Omron CX-Programmer project NewProject (CX-Programmer 9.73)

# PLC NewPLC1: CP1L-E EM

## Global symbols (name address type ; comment)
0.00 BOOL  ; passo a passo formador fila entrada roler 41
0.01 BOOL  ; sensor peças maquineta descarga 41
0.02 BOOL  ; sensor sobre rolos entrada forno
0.03 BOOL  ; rele espaco forno 17 (saida 3.03)
0.04 BOOL  ; passo a passo formador fila entrada roler 42
0.05 BOOL  ; status roller desc. 42
0.06 BOOL  ; bancalino baixo carga forno 18
0.07 BOOL  ; rele forno 18 (saida 3.03)
0.08 BOOL  ; cnt de planos de carga 43
0.09 BOOL  ; cnt de planos de descarga 43
0.10 BOOL  ; bancalino entrada forno
0.11 BOOL  ; rele forno 22
1.00 BOOL  ; contagem de planos da carga carro
1.01 BOOL  ; status roller C41
1.02 BOOL  ; contador de gavetas carga roller mf42
1.03 BOOL  ; status roller C41
1.04 BOOL  ; contador descarga gaveta roller descarga mf42
1.05 BOOL  ; contagem de planos da descarga carro
1.08 BOOL  ; contagem peças roller carga 43
1.09 BOOL  ; status roller C43
1.11 BOOL  ; status roller D43
20.00 BOOL  ; reset retorno peças
20.01 BOOL  ; reset retorno peças
20.02 BOOL  ; reset retorno peças
30.02 BOOL  ; estoque vazio
30.04 BOOL  ; estoque zero mf42
30.05 BOOL  ; comparador planos  vazios
50.00 BOOL  ; liga cnt10
50.01 BOOL  ; reset cnt10
50.02 BOOL  ; liga cnt11
50.03 BOOL  ; reset cnt11
50.04 BOOL  ; liga cnt12
50.05 BOOL  ; reset cnt12
C0010 BOOL  ; reset inicio turno 1
C0011 BOOL  ; reset inicio turno 2
C0012 BOOL  ; reset inicio turno 3
C43 CHANNEL  ; contador de planos da 43
D1 CHANNEL  ; contador peças
D107 CHANNEL  ; peças por fila entrada forno
D205 CHANNEL  ; Segundos Relógio
D206 CHANNEL  ; Minutos Relógio
D207 CHANNEL  ; Horas Relogio
D208 CHANNEL  ; Dia Relógio
D209 CHANNEL  ; Mes Relogio
D210 CHANNEL  ; Ano Relogio
D211 CHANNEL  ; Ano Relogio 4 Digitos
D300 CHANNEL  ; Ano Relógio
D3001 CHANNEL  ; receita de destino RC43
D301 CHANNEL  ; Ano Relógio 4 digitos
D3800 CHANNEL  ; receita de destino F22
D400 CHANNEL  ; dia do mes
D402 CHANNEL  ; primeiro DM de contagem forno
D404 CHANNEL  ; peças por fila f17
D406 CHANNEL  ; peças por fila f18
D408 CHANNEL  ; peças por fila f22
D410 CHANNEL  ; primeiro DM envio roller
D500 CHANNEL  ; turno 1,2,3
D800 CHANNEL  ; horas
D802 CHANNEL  ; minutos
D804 CHANNEL  ; segundos
D806 CHANNEL  ; dia calendario
D808 CHANNEL  ; mês calendario
D810 CHANNEL  ; mês selecionado
D811 CHANNEL  ; linha selecionada
D910 CHANNEL  ; mês selecionado
H10.00 BOOL  ; forno com espaço
H10.01 BOOL  ; status roller carga 41
H10.02 BOOL  ; forno com espaço
H10.03 BOOL  ; roller carga 42
H10.04 BOOL  ; forno com espaço
H10.05 BOOL  ; status roller descarga 42
H10.06 BOOL  ; roller descarga 41
H10.07 BOOL  ; roller carga 43
H10.08 BOOL  ; status roller descarga 43
H19.15 BOOL  ; correção estoque IHM (mais)
H20.00 BOOL  ; Envia relogio superviório
H20.01 BOOL  ; correção estoque IHM (menos)
H20.02 BOOL  ; correção estoque IHM (menos)
H20.03 BOOL  ; correção estoque IHM (mais)
H20.04 BOOL  ; correção estoque IHM (menos)
H20.05 BOOL  ; correção estoque IHM (mais)
H20.06 BOOL  ; correcão estoque(menos)
H20.07 BOOL  ; correcão estoque(mais)
H20.08 BOOL  ; correcão estoque(menos)
H20.09 BOOL  ; correcão estoque(mais)
H20.10 BOOL  ; correcão estoque(menos)
H20.11 BOOL  ; correcão estoque(mais)
H30.00 BOOL  ; inicia contagem turno 1
H30.01 BOOL  ; inicia contagem turno 2
H30.02 BOOL  ; iniio contagem turno 3
T0001 BOOL  ; filtro senso
Banco_de_Dados Contador_de_Peças_RC43
Banco_de_Dados_ Contador_de_Peças_RC42
Banco_de_Dados_F17 Contador_de_Peças_F17
Banco_de_Dados_F18 Contador_de_Peças_F18
Banco_de_Dados_F22 Contador_de_Peças_F22
Banco_de_Dados_R42 Contador_de_Peças_RC42
Banco_de_Dados_R43 Contador_de_Peças_RC43
Banco_de_dados Contador_de_Peças_RC41
Banco_de_dados_R41 Contador_de_Peças_RC41
Reservado_1 D300 CHANNEL  ; reservado para elipse
Reservado_10 D309 CHANNEL  ; reservado para elipse
Reservado_11 D310 CHANNEL  ; reservado para elipse
Reservado_2 D301 CHANNEL  ; reservado para elipse
Reservado_3 D302 CHANNEL  ; reservado para elipse
Reservado_4 D303 CHANNEL  ; reservado para elipse
Reservado_5 D304 CHANNEL  ; reservado para elipse
Reservado_6 D305 CHANNEL  ; reservado para elipse
Reservado_7 D306 CHANNEL  ; reservado para elipse
Reservado_8 D307 CHANNEL  ; reservado para elipse
Reservado_9 D308 CHANNEL  ; reservado para elipse

## Program NewProgram1 (cyclic task 0)

### Section Principal

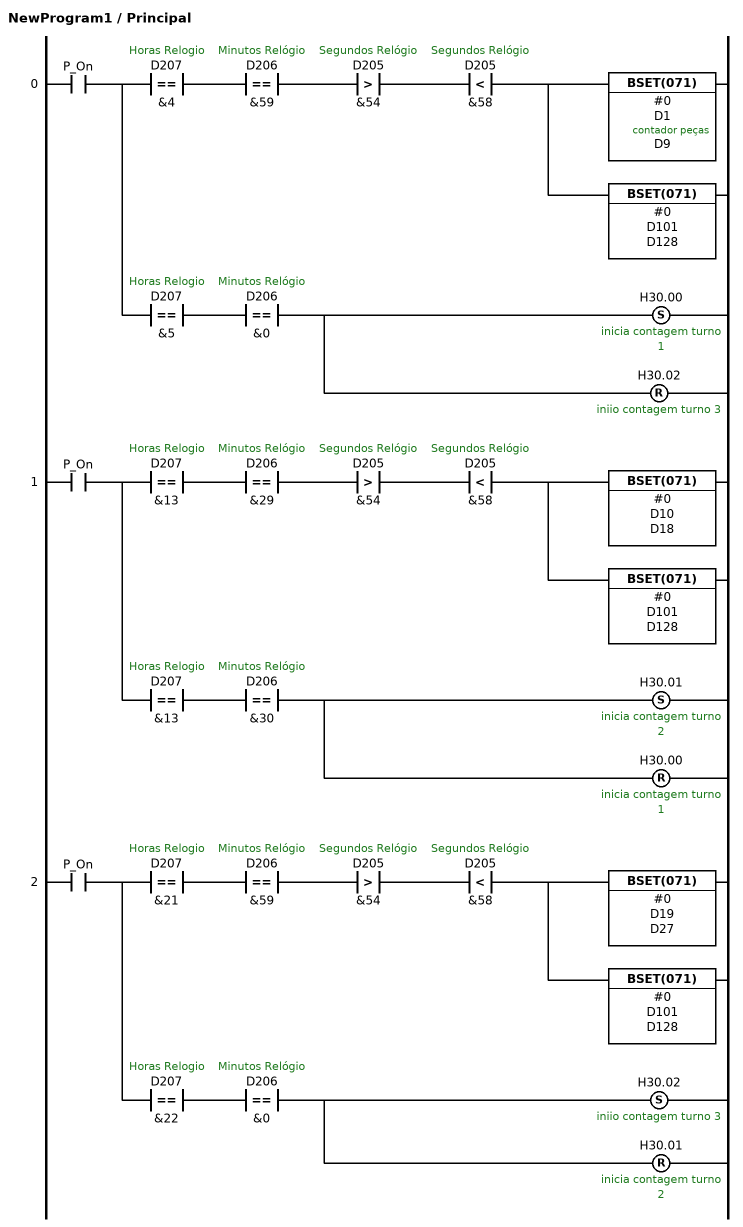
; rung 0
LD P_On
OUT TR0
AND=(300) D207 &4  ; Horas Relogio
AND=(300) D206 &59  ; Minutos Relógio
AND>(320) D205 &54  ; Segundos Relógio
AND<(310) D205 &58  ; Segundos Relógio
BSET(071) #0 D1 D9  ; contador peças
BSET(071) #0 D101 D128
LD TR0
AND=(300) D207 &5  ; Horas Relogio
AND=(300) D206 &0  ; Minutos Relógio
SET H30.00  ; inicia contagem turno 1
RSET H30.02  ; iniio contagem turno 3
; rung 1
LD P_On
OUT TR0
AND=(300) D207 &13  ; Horas Relogio
AND=(300) D206 &29  ; Minutos Relógio
AND>(320) D205 &54  ; Segundos Relógio
AND<(310) D205 &58  ; Segundos Relógio
BSET(071) #0 D10 D18
BSET(071) #0 D101 D128
LD TR0
AND=(300) D207 &13  ; Horas Relogio
AND=(300) D206 &30  ; Minutos Relógio
SET H30.01  ; inicia contagem turno 2
RSET H30.00  ; inicia contagem turno 1
; rung 2
LD P_On
OUT TR0
AND=(300) D207 &21  ; Horas Relogio
AND=(300) D206 &59  ; Minutos Relógio
AND>(320) D205 &54  ; Segundos Relógio
AND<(310) D205 &58  ; Segundos Relógio
BSET(071) #0 D19 D27
BSET(071) #0 D101 D128
LD TR0
AND=(300) D207 &22  ; Horas Relogio
AND=(300) D206 &0  ; Minutos Relógio
SET H30.02  ; iniio contagem turno 3
RSET H30.01  ; inicia contagem turno 2

### Section MF41

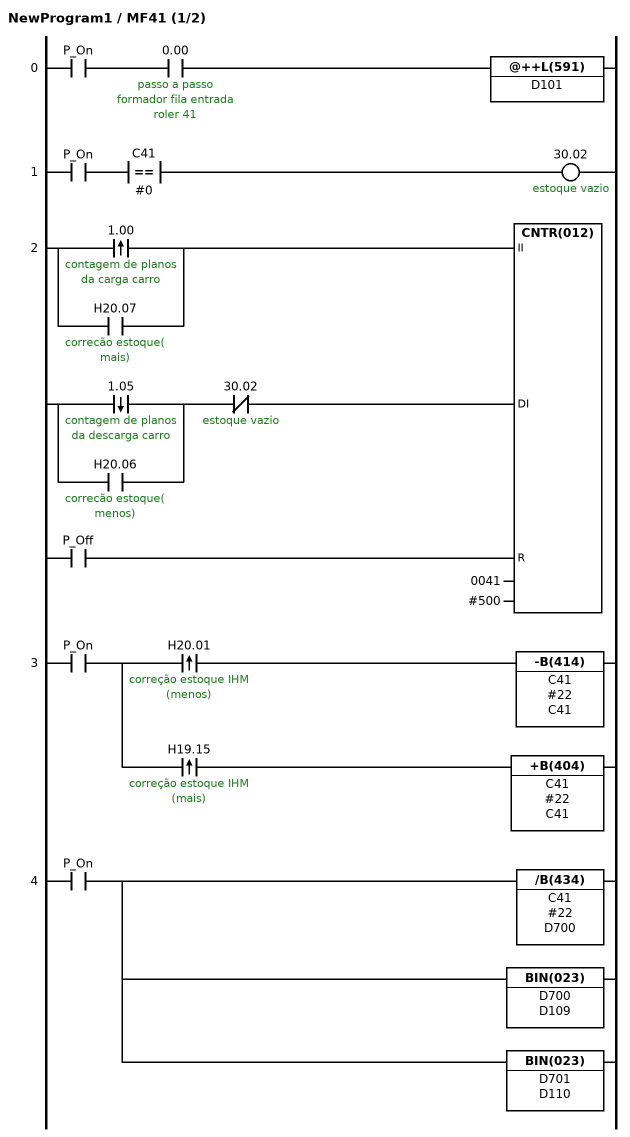
; rung 0
LD P_On
AND 0.00  ; passo a passo formador fila entrada roler 41
@++L(591) D101
; rung 1
LD P_On
AND=(300) C41 #0
OUT 30.02  ; estoque vazio
; rung 2
@LD 1.00  ; contagem de planos da carga carro
OR H20.07  ; correcão estoque(mais)
%LD 1.05  ; contagem de planos da descarga carro
OR H20.06  ; correcão estoque(menos)
ANDNOT 30.02  ; estoque vazio
LD P_Off
CNTR(012) 0041 #500
; rung 3
LD P_On
OUT TR0
@AND H20.01  ; correção estoque IHM (menos)
-B(414) C41 #22 C41
LD TR0
@AND H19.15  ; correção estoque IHM (mais)
+B(404) C41 #22 C41
; rung 4
LD P_On
/B(434) C41 #22 D700
BIN(023) D700 D109
BIN(023) D701 D110

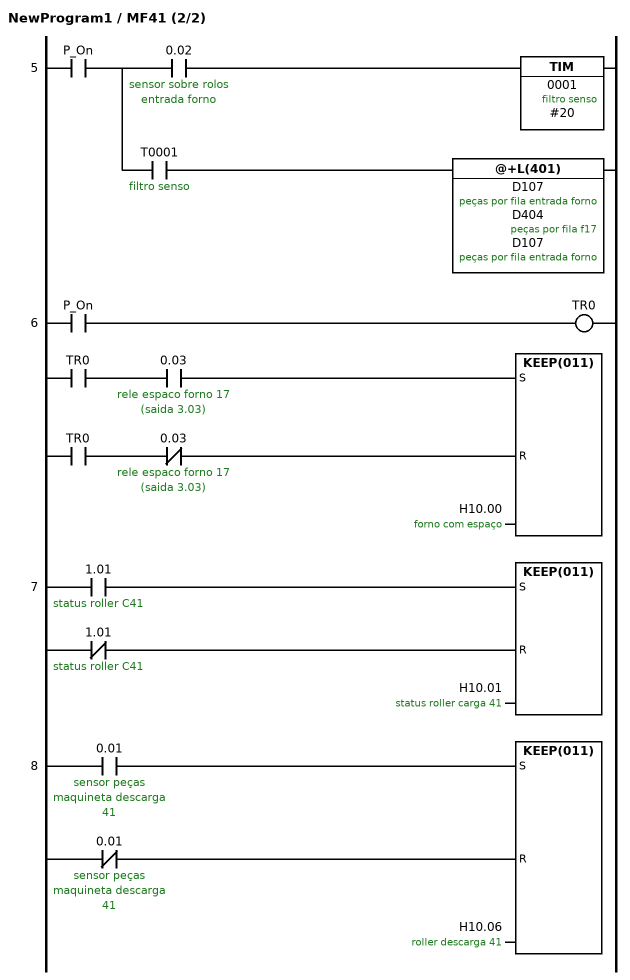
; rung 5
LD P_On
OUT TR0
AND 0.02  ; sensor sobre rolos entrada forno
TIM 0001 #20  ; filtro senso
LD TR0
AND T0001  ; filtro senso
@+L(401) D107 D404 D107  ; peças por fila entrada forno, peças por fila f17
; rung 6
LD P_On
OUT TR0
AND 0.03  ; rele espaco forno 17 (saida 3.03)
LD TR0
ANDNOT 0.03  ; rele espaco forno 17 (saida 3.03)
KEEP(011) H10.00  ; forno com espaço
; rung 7
LD 1.01  ; status roller C41
LDNOT 1.01  ; status roller C41
KEEP(011) H10.01  ; status roller carga 41
; rung 8
LD 0.01  ; sensor peças maquineta descarga 41
LDNOT 0.01  ; sensor peças maquineta descarga 41
KEEP(011) H10.06  ; roller descarga 41

### Section MF42

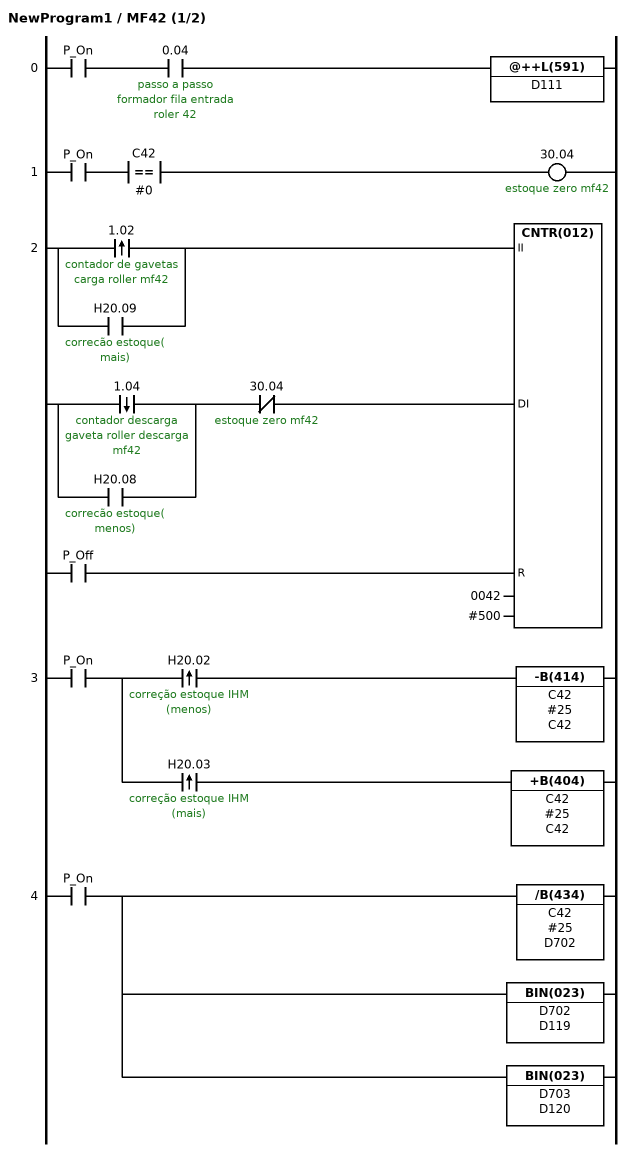
; rung 0
LD P_On
AND 0.04  ; passo a passo formador fila entrada roler 42
@++L(591) D111
; rung 1
LD P_On
AND=(300) C42 #0
OUT 30.04  ; estoque zero mf42
; rung 2
@LD 1.02  ; contador de gavetas carga roller mf42
OR H20.09  ; correcão estoque(mais)
%LD 1.04  ; contador descarga gaveta roller descarga mf42
OR H20.08  ; correcão estoque(menos)
ANDNOT 30.04  ; estoque zero mf42
LD P_Off
CNTR(012) 0042 #500
; rung 3
LD P_On
OUT TR0
@AND H20.02  ; correção estoque IHM (menos)
-B(414) C42 #25 C42
LD TR0
@AND H20.03  ; correção estoque IHM (mais)
+B(404) C42 #25 C42
; rung 4
LD P_On
/B(434) C42 #25 D702
BIN(023) D702 D119
BIN(023) D703 D120

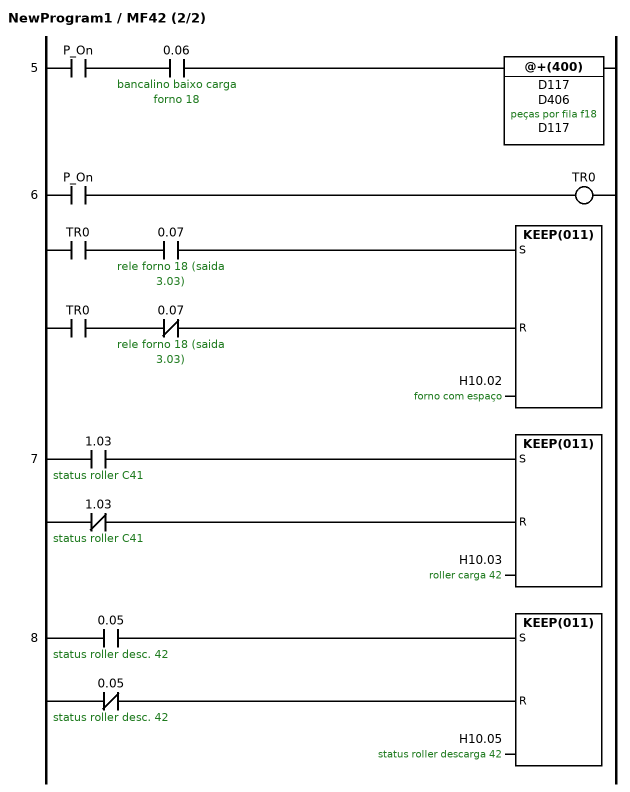
; rung 5
LD P_On
AND 0.06  ; bancalino baixo carga forno 18
@+(400) D117 D406 D117  ; peças por fila f18
; rung 6
LD P_On
OUT TR0
AND 0.07  ; rele forno 18 (saida 3.03)
LD TR0
ANDNOT 0.07  ; rele forno 18 (saida 3.03)
KEEP(011) H10.02  ; forno com espaço
; rung 7
LD 1.03  ; status roller C41
LDNOT 1.03  ; status roller C41
KEEP(011) H10.03  ; roller carga 42
; rung 8
LD 0.05  ; status roller desc. 42
LDNOT 0.05  ; status roller desc. 42
KEEP(011) H10.05  ; status roller descarga 42

### Section MF43

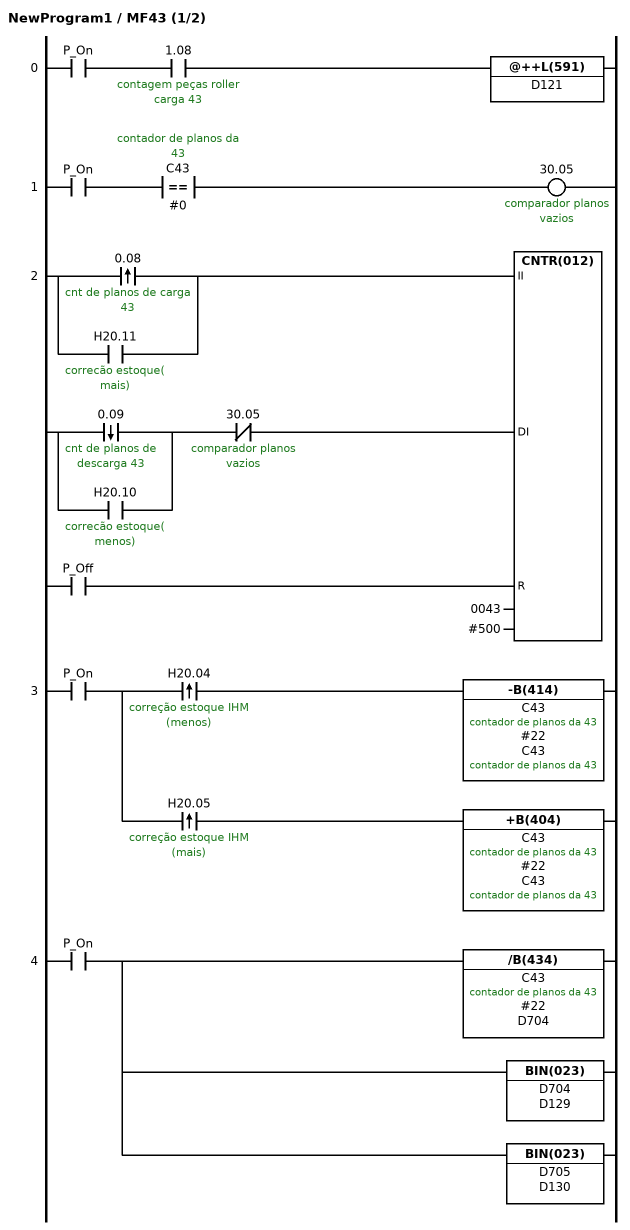
; rung 0
LD P_On
AND 1.08  ; contagem peças roller carga 43
@++L(591) D121
; rung 1
LD P_On
AND=(300) C43 #0  ; contador de planos da 43
OUT 30.05  ; comparador planos  vazios
; rung 2
@LD 0.08  ; cnt de planos de carga 43
OR H20.11  ; correcão estoque(mais)
%LD 0.09  ; cnt de planos de descarga 43
OR H20.10  ; correcão estoque(menos)
ANDNOT 30.05  ; comparador planos  vazios
LD P_Off
CNTR(012) 0043 #500
; rung 3
LD P_On
OUT TR0
@AND H20.04  ; correção estoque IHM (menos)
-B(414) C43 #22 C43  ; contador de planos da 43
LD TR0
@AND H20.05  ; correção estoque IHM (mais)
+B(404) C43 #22 C43  ; contador de planos da 43
; rung 4
LD P_On
/B(434) C43 #22 D704  ; contador de planos da 43
BIN(023) D704 D129
BIN(023) D705 D130

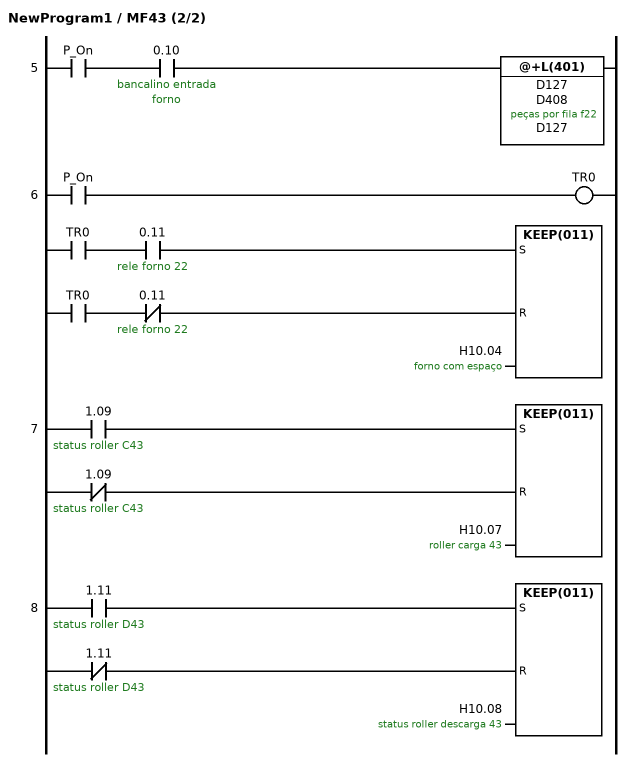
; rung 5
LD P_On
AND 0.10  ; bancalino entrada forno
@+L(401) D127 D408 D127  ; peças por fila f22
; rung 6
LD P_On
OUT TR0
AND 0.11  ; rele forno 22
LD TR0
ANDNOT 0.11  ; rele forno 22
KEEP(011) H10.04  ; forno com espaço
; rung 7
LD 1.09  ; status roller C43
LDNOT 1.09  ; status roller C43
KEEP(011) H10.07  ; roller carga 43
; rung 8
LD 1.11  ; status roller D43
LDNOT 1.11  ; status roller D43
KEEP(011) H10.08  ; status roller descarga 43

### Section MF41_ESPAÇO

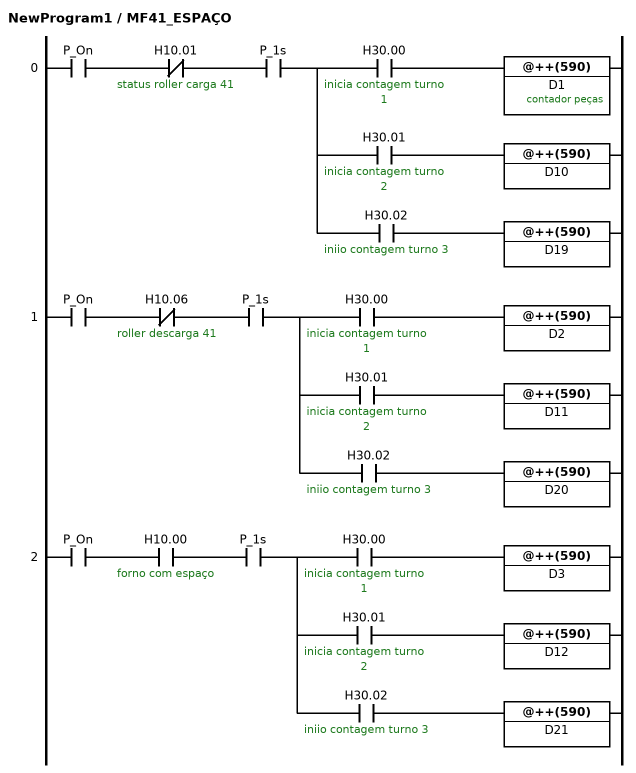
; rung 0
LD P_On
ANDNOT H10.01  ; status roller carga 41
AND P_1s
OUT TR0
AND H30.00  ; inicia contagem turno 1
@++(590) D1  ; contador peças  // 
LD TR0
AND H30.01  ; inicia contagem turno 2
@++(590) D10  // 
LD TR0
AND H30.02  ; iniio contagem turno 3
@++(590) D19  // 
; rung 1
LD P_On
ANDNOT H10.06  ; roller descarga 41
AND P_1s
OUT TR0
AND H30.00  ; inicia contagem turno 1
@++(590) D2  // 
LD TR0
AND H30.01  ; inicia contagem turno 2
@++(590) D11  // 
LD TR0
AND H30.02  ; iniio contagem turno 3
@++(590) D20  // 
; rung 2
LD P_On
AND H10.00  ; forno com espaço
AND P_1s
OUT TR0
AND H30.00  ; inicia contagem turno 1
@++(590) D3  // 
LD TR0
AND H30.01  ; inicia contagem turno 2
@++(590) D12  // 
LD TR0
AND H30.02  ; iniio contagem turno 3
@++(590) D21  // 

### Section MF42_ESPAÇO

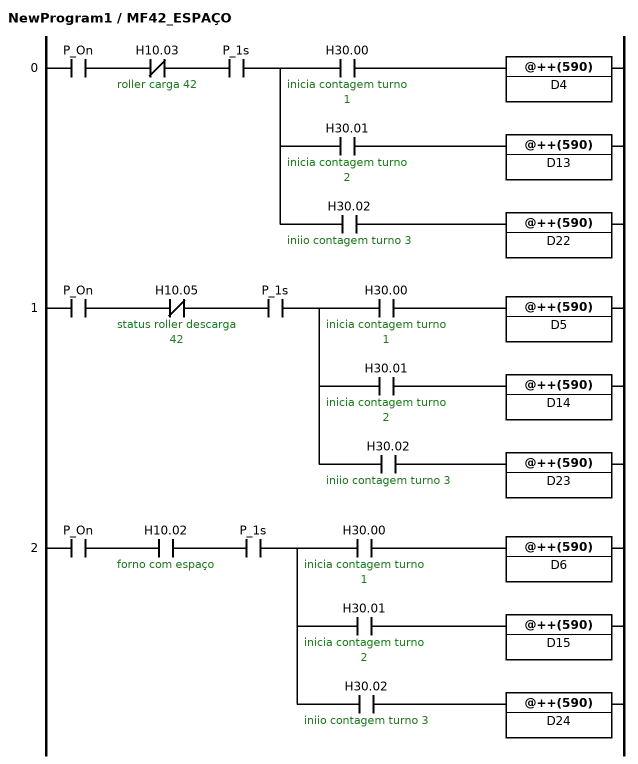
; rung 0
LD P_On
ANDNOT H10.03  ; roller carga 42
AND P_1s
OUT TR0
AND H30.00  ; inicia contagem turno 1
@++(590) D4  // 
LD TR0
AND H30.01  ; inicia contagem turno 2
@++(590) D13  // 
LD TR0
AND H30.02  ; iniio contagem turno 3
@++(590) D22  // 
; rung 1
LD P_On
ANDNOT H10.05  ; status roller descarga 42
AND P_1s
OUT TR0
AND H30.00  ; inicia contagem turno 1
@++(590) D5  // 
LD TR0
AND H30.01  ; inicia contagem turno 2
@++(590) D14  // 
LD TR0
AND H30.02  ; iniio contagem turno 3
@++(590) D23  // 
; rung 2
LD P_On
AND H10.02  ; forno com espaço
AND P_1s
OUT TR0
AND H30.00  ; inicia contagem turno 1
@++(590) D6  // 
LD TR0
AND H30.01  ; inicia contagem turno 2
@++(590) D15  // 
LD TR0
AND H30.02  ; iniio contagem turno 3
@++(590) D24  // 

### Section MF43_ESPAÇO

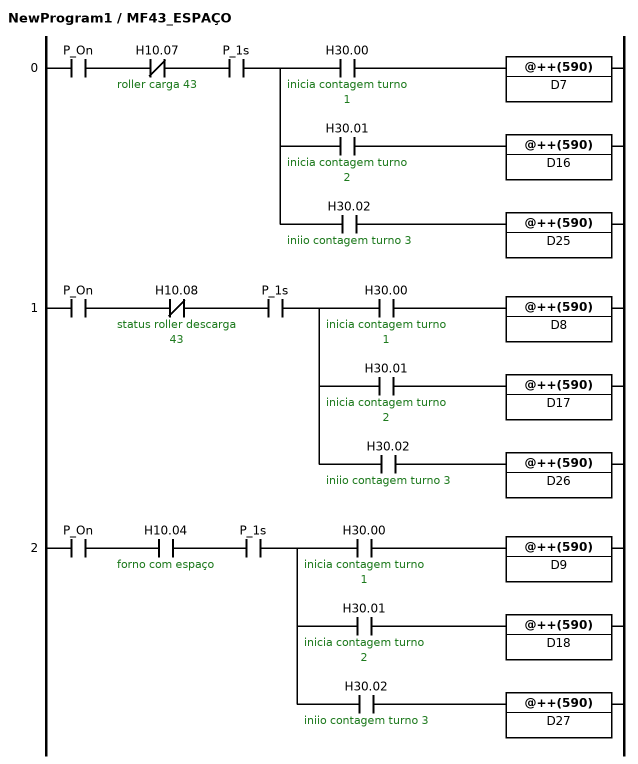
; rung 0
LD P_On
ANDNOT H10.07  ; roller carga 43
AND P_1s
OUT TR0
AND H30.00  ; inicia contagem turno 1
@++(590) D7  // 
LD TR0
AND H30.01  ; inicia contagem turno 2
@++(590) D16  // 
LD TR0
AND H30.02  ; iniio contagem turno 3
@++(590) D25  // 
; rung 1
LD P_On
ANDNOT H10.08  ; status roller descarga 43
AND P_1s
OUT TR0
AND H30.00  ; inicia contagem turno 1
@++(590) D8  // 
LD TR0
AND H30.01  ; inicia contagem turno 2
@++(590) D17  // 
LD TR0
AND H30.02  ; iniio contagem turno 3
@++(590) D26  // 
; rung 2
LD P_On
AND H10.04  ; forno com espaço
AND P_1s
OUT TR0
AND H30.00  ; inicia contagem turno 1
@++(590) D9  // 
LD TR0
AND H30.01  ; inicia contagem turno 2
@++(590) D18  // 
LD TR0
AND H30.02  ; iniio contagem turno 3
@++(590) D27  // 

### Section Banco_de_Dados

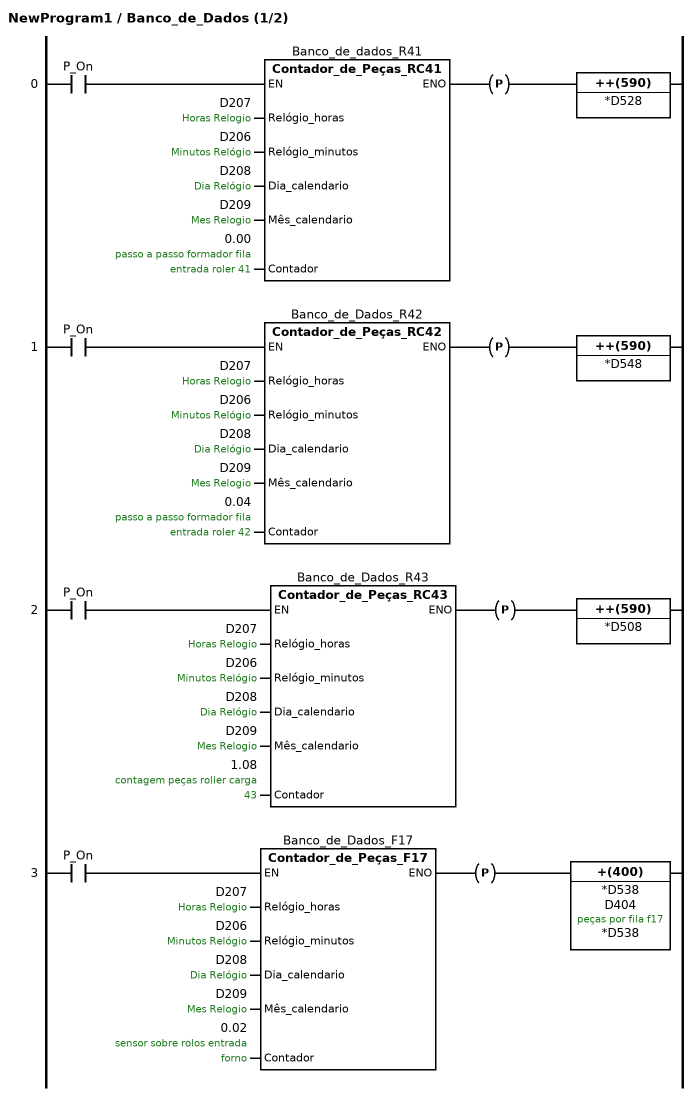
; rung 0
LD P_On
CALL Banco_de_dados_R41 : Contador_de_Peças_RC41 (Relógio_horas := D207, Relógio_minutos := D206, Dia_calendario := D208, Mês_calendario := D209, Contador := 0.00)  ; Horas Relogio, Minutos Relógio, Dia Relógio, Mes Relogio, passo a passo formador fila entrada roler 41
UP(521)
++(590) *D528
; rung 1
LD P_On
CALL Banco_de_Dados_R42 : Contador_de_Peças_RC42 (Relógio_horas := D207, Relógio_minutos := D206, Dia_calendario := D208, Mês_calendario := D209, Contador := 0.04)  ; Horas Relogio, Minutos Relógio, Dia Relógio, Mes Relogio, passo a passo formador fila entrada roler 42
UP(521)
++(590) *D548
; rung 2
LD P_On
CALL Banco_de_Dados_R43 : Contador_de_Peças_RC43 (Relógio_horas := D207, Relógio_minutos := D206, Dia_calendario := D208, Mês_calendario := D209, Contador := 1.08)  ; Horas Relogio, Minutos Relógio, Dia Relógio, Mes Relogio, contagem peças roller carga 43
UP(521)
++(590) *D508
; rung 3
LD P_On
CALL Banco_de_Dados_F17 : Contador_de_Peças_F17 (Relógio_horas := D207, Relógio_minutos := D206, Dia_calendario := D208, Mês_calendario := D209, Contador := 0.02)  ; Horas Relogio, Minutos Relógio, Dia Relógio, Mes Relogio, sensor sobre rolos entrada forno
UP(521)
+(400) *D538 D404 *D538  ; peças por fila f17

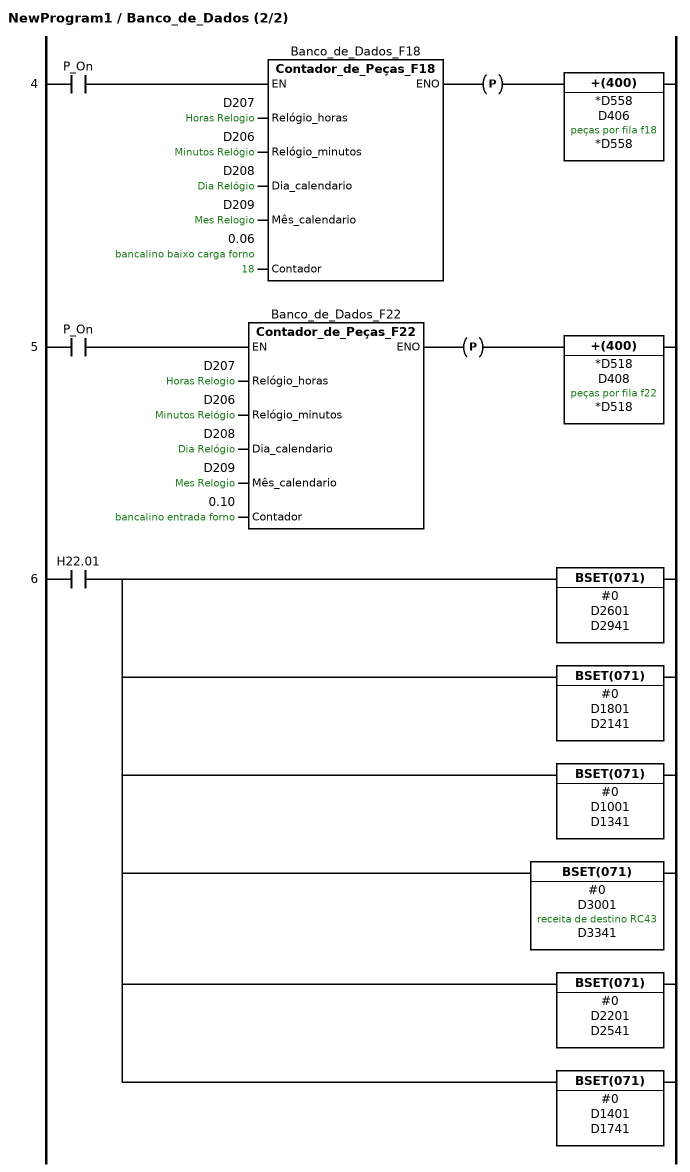
; rung 4
LD P_On
CALL Banco_de_Dados_F18 : Contador_de_Peças_F18 (Relógio_horas := D207, Relógio_minutos := D206, Dia_calendario := D208, Mês_calendario := D209, Contador := 0.06)  ; Horas Relogio, Minutos Relógio, Dia Relógio, Mes Relogio, bancalino baixo carga forno 18
UP(521)
+(400) *D558 D406 *D558  ; peças por fila f18
; rung 5
LD P_On
CALL Banco_de_Dados_F22 : Contador_de_Peças_F22 (Relógio_horas := D207, Relógio_minutos := D206, Dia_calendario := D208, Mês_calendario := D209, Contador := 0.10)  ; Horas Relogio, Minutos Relógio, Dia Relógio, Mes Relogio, bancalino entrada forno
UP(521)
+(400) *D518 D408 *D518  ; peças por fila f22
; rung 6
LD H22.01
BSET(071) #0 D2601 D2941
BSET(071) #0 D1801 D2141
BSET(071) #0 D1001 D1341
BSET(071) #0 D3001 D3341  ; receita de destino RC43
BSET(071) #0 D2201 D2541
BSET(071) #0 D1401 D1741

### Section Transferencia_excel

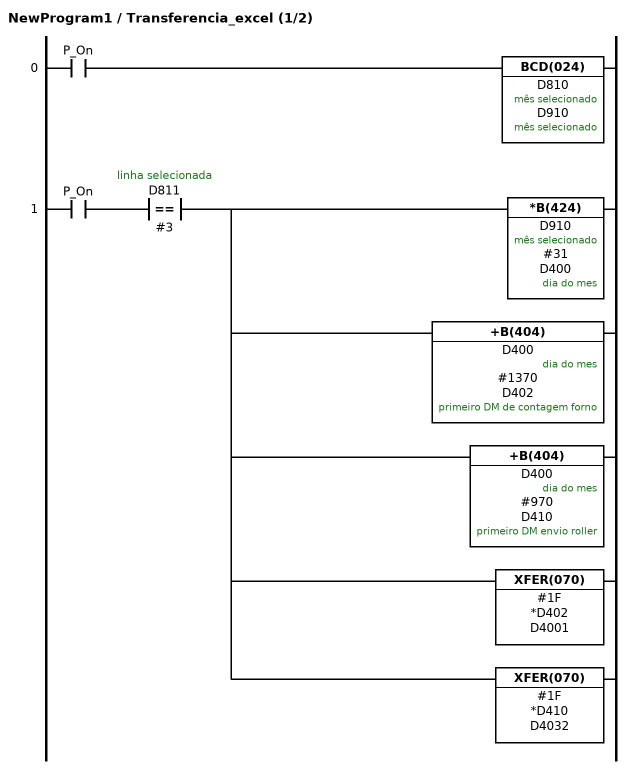
; rung 0
LD P_On
BCD(024) D810 D910  ; mês selecionado
; rung 1
LD P_On
AND=(300) D811 #3  ; linha selecionada
*B(424) D910 #31 D400  ; mês selecionado, dia do mes
+B(404) D400 #1370 D402  ; dia do mes, primeiro DM de contagem forno
+B(404) D400 #970 D410  ; dia do mes, primeiro DM envio roller
XFER(070) #1F *D402 D4001
XFER(070) #1F *D410 D4032

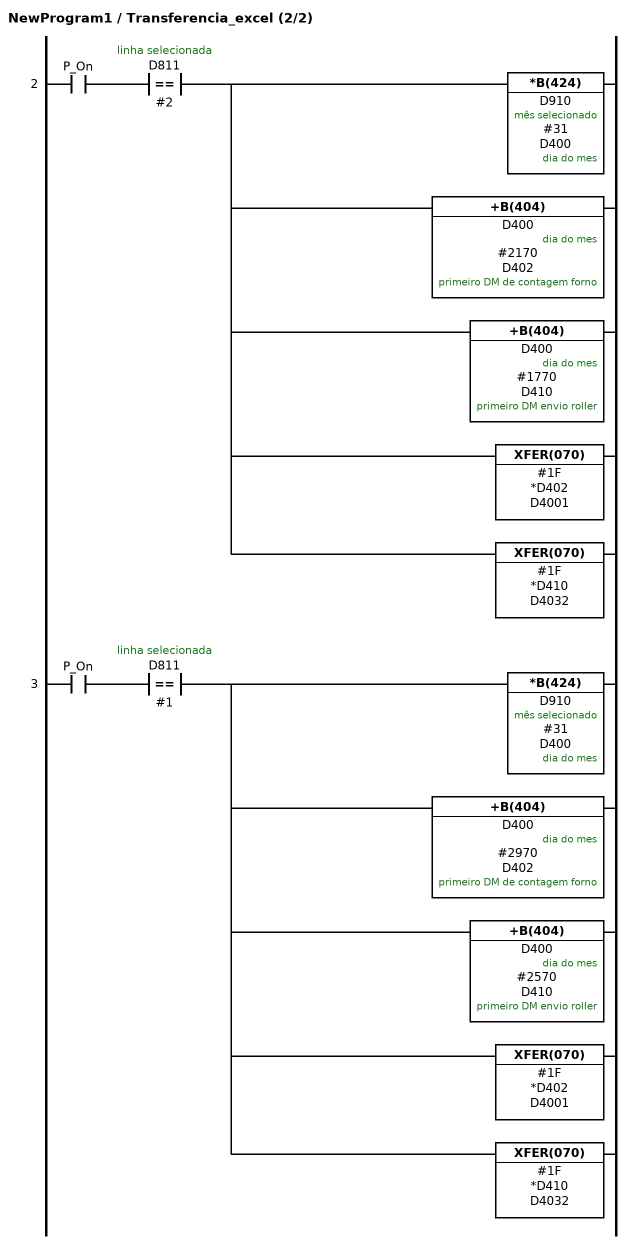
; rung 2
LD P_On
AND=(300) D811 #2  ; linha selecionada
*B(424) D910 #31 D400  ; mês selecionado, dia do mes
+B(404) D400 #2170 D402  ; dia do mes, primeiro DM de contagem forno
+B(404) D400 #1770 D410  ; dia do mes, primeiro DM envio roller
XFER(070) #1F *D402 D4001
XFER(070) #1F *D410 D4032
; rung 3
LD P_On
AND=(300) D811 #1  ; linha selecionada
*B(424) D910 #31 D400  ; mês selecionado, dia do mes
+B(404) D400 #2970 D402  ; dia do mes, primeiro DM de contagem forno
+B(404) D400 #2570 D410  ; dia do mes, primeiro DM envio roller
XFER(070) #1F *D402 D4001
XFER(070) #1F *D410 D4032

### Section Relogio

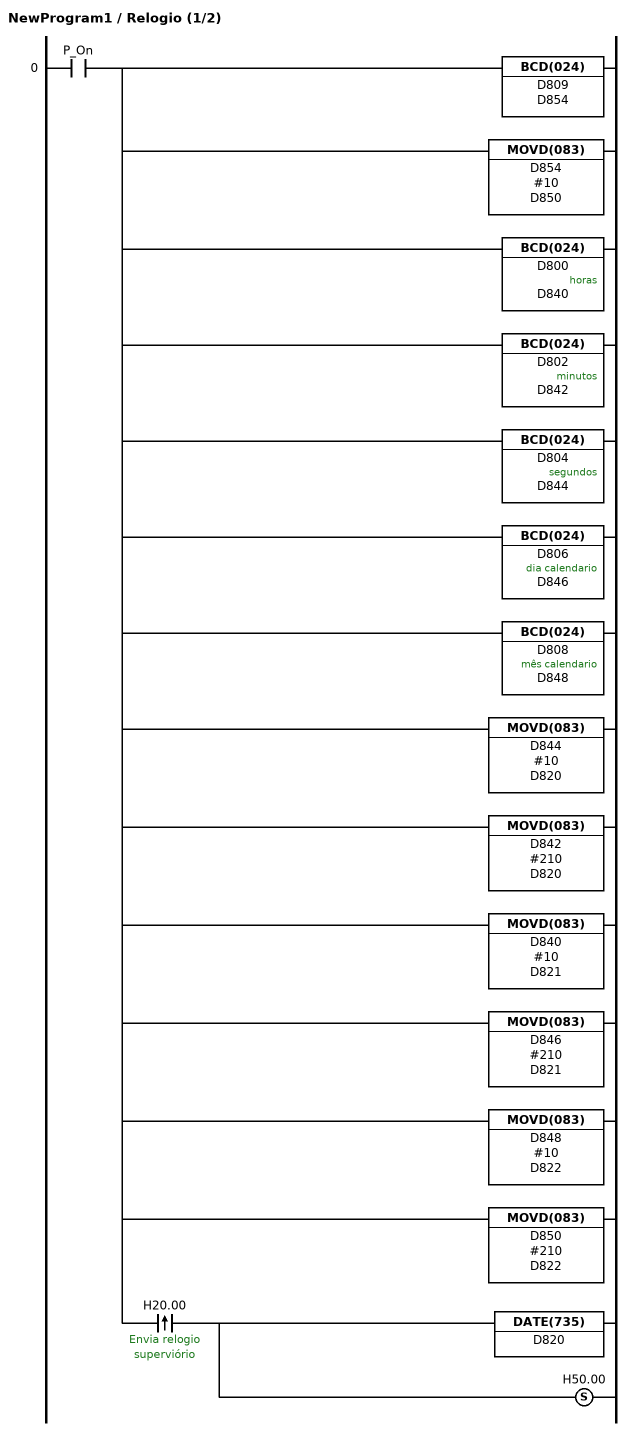
; rung 0
LD P_On
BCD(024) D809 D854
MOVD(083) D854 #10 D850
BCD(024) D800 D840  ; horas
BCD(024) D802 D842  ; minutos
BCD(024) D804 D844  ; segundos
BCD(024) D806 D846  ; dia calendario
BCD(024) D808 D848  ; mês calendario
MOVD(083) D844 #10 D820
MOVD(083) D842 #210 D820
MOVD(083) D840 #10 D821
MOVD(083) D846 #210 D821
MOVD(083) D848 #10 D822
MOVD(083) D850 #210 D822
@AND H20.00  ; Envia relogio superviório
DATE(735) D820
SET H50.00

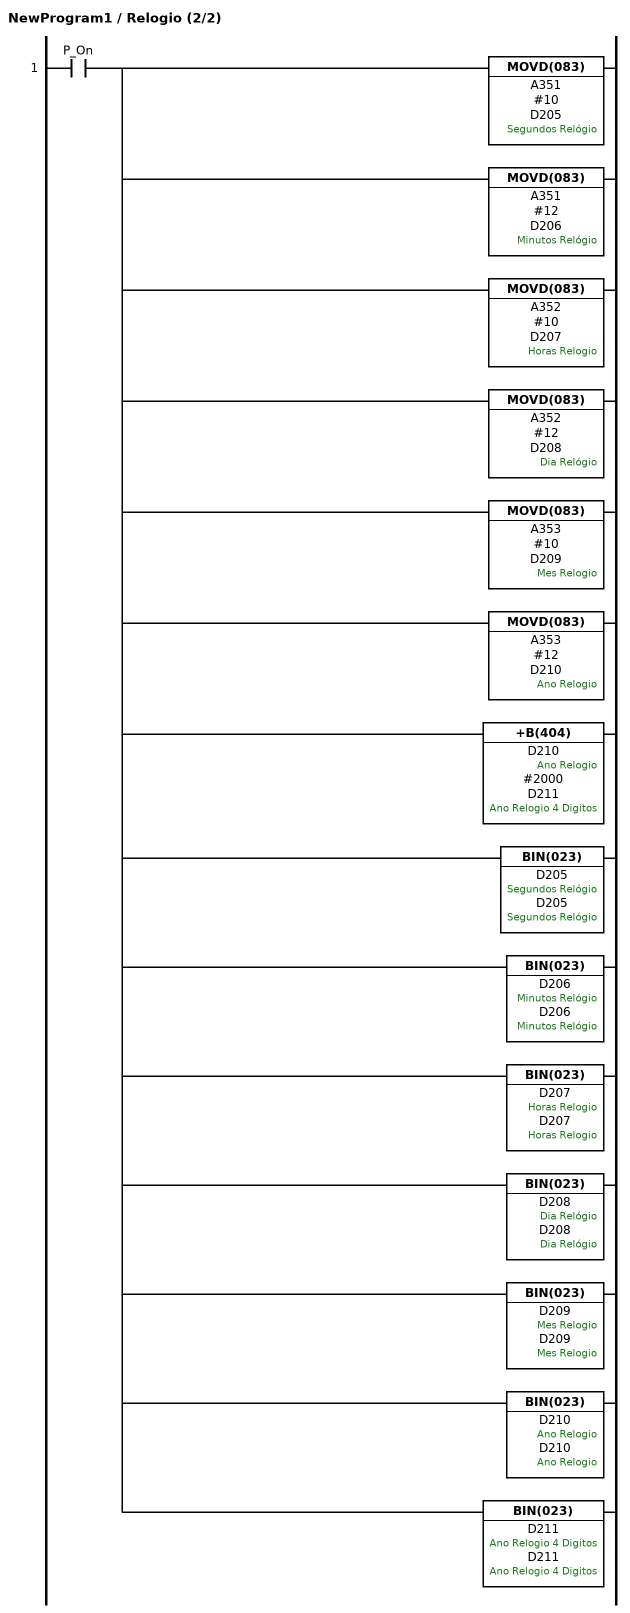
; rung 1
LD P_On
MOVD(083) A351 #10 D205  ; Segundos Relógio
MOVD(083) A351 #12 D206  ; Minutos Relógio
MOVD(083) A352 #10 D207  ; Horas Relogio
MOVD(083) A352 #12 D208  ; Dia Relógio
MOVD(083) A353 #10 D209  ; Mes Relogio
MOVD(083) A353 #12 D210  ; Ano Relogio
+B(404) D210 #2000 D211  ; Ano Relogio, Ano Relogio 4 Digitos
BIN(023) D205 D205  ; Segundos Relógio
BIN(023) D206 D206  ; Minutos Relógio
BIN(023) D207 D207  ; Horas Relogio
BIN(023) D208 D208  ; Dia Relógio
BIN(023) D209 D209  ; Mes Relogio
BIN(023) D210 D210  ; Ano Relogio
BIN(023) D211 D211  ; Ano Relogio 4 Digitos

### Section End
; rung 0
END(001)

## Function block Contador_de_Peças_F17
VAR_INPUT
  Relógio_horas : WORD;
  Relógio_minutos : WORD;
  Dia_calendario : WORD;
  Mês_calendario : WORD;
  Contador : BOOL;
END_VAR
VAR
  _31dias_vezes_2 AT D530 : WORD;
  Ponteiro_DWord AT D532 : WORD;
  Memória_de_Armazenagem AT D534 : WORD;
  Memoria_contagem_BIN AT D536 : WORD;
  Memoria_contagem_BCD AT D538 : WORD;
END_VAR

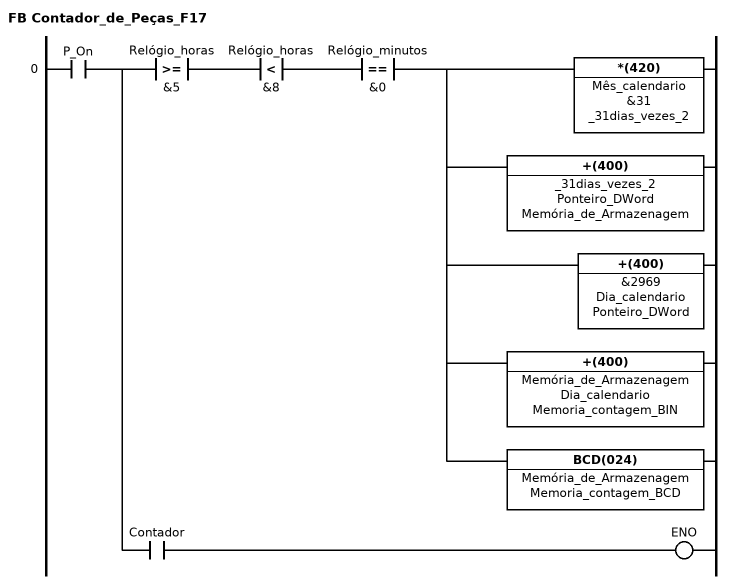
; rung 0
LD P_On
OUT TR0
AND>=(325) Relógio_horas &5
AND<(310) Relógio_horas &8
AND=(300) Relógio_minutos &0
*(420) Mês_calendario &31 _31dias_vezes_2
+(400) _31dias_vezes_2 Ponteiro_DWord Memória_de_Armazenagem
+(400) &2969 Dia_calendario Ponteiro_DWord
+(400) Memória_de_Armazenagem Dia_calendario Memoria_contagem_BIN
BCD(024) Memória_de_Armazenagem Memoria_contagem_BCD
LD TR0
AND Contador
OUT ENO

## Function block Contador_de_Peças_F18
VAR_INPUT
  Relógio_horas : WORD;
  Relógio_minutos : WORD;
  Dia_calendario : WORD;
  Mês_calendario : WORD;
  Contador : BOOL;
END_VAR
VAR
  _31dias_vezes_2 AT D550 : WORD;
  Ponteiro_DWord AT D552 : WORD;
  Memória_de_Armazenagem AT D554 : WORD;
  Memoria_contagem_BIN AT D556 : WORD;
  Memoria_contagem_BCD AT D558 : WORD;
END_VAR

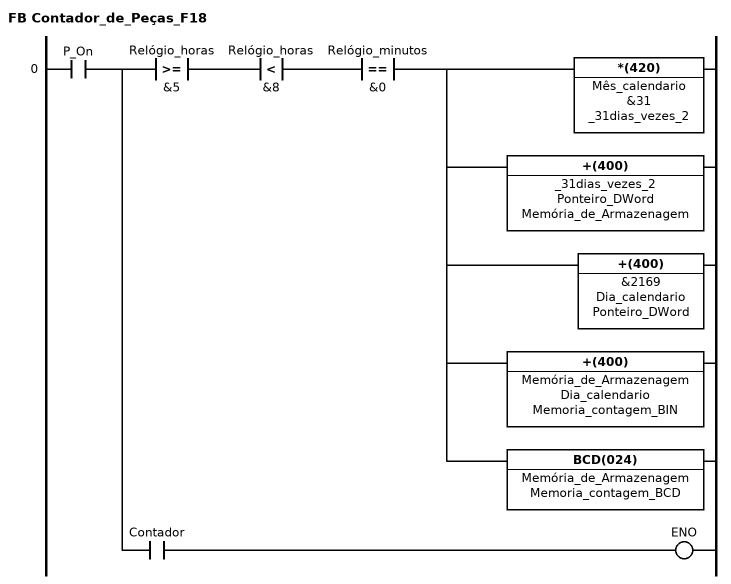
; rung 0
LD P_On
OUT TR0
AND>=(325) Relógio_horas &5
AND<(310) Relógio_horas &8
AND=(300) Relógio_minutos &0
*(420) Mês_calendario &31 _31dias_vezes_2
+(400) _31dias_vezes_2 Ponteiro_DWord Memória_de_Armazenagem
+(400) &2169 Dia_calendario Ponteiro_DWord
+(400) Memória_de_Armazenagem Dia_calendario Memoria_contagem_BIN
BCD(024) Memória_de_Armazenagem Memoria_contagem_BCD
LD TR0
AND Contador
OUT ENO

## Function block Contador_de_Peças_F22
VAR_INPUT
  Relógio_horas : WORD;
  Relógio_minutos : WORD;
  Dia_calendario : WORD;
  Mês_calendario : WORD;
  Contador : BOOL;
END_VAR
VAR
  _31dias_vezes_2 AT D510 : WORD;
  Ponteiro_DWord AT D512 : WORD;
  Memória_de_Armazenagem AT D514 : WORD;
  Memoria_contagem_BIN AT D516 : WORD;
  Memoria_contagem_BCD AT D518 : WORD;
END_VAR

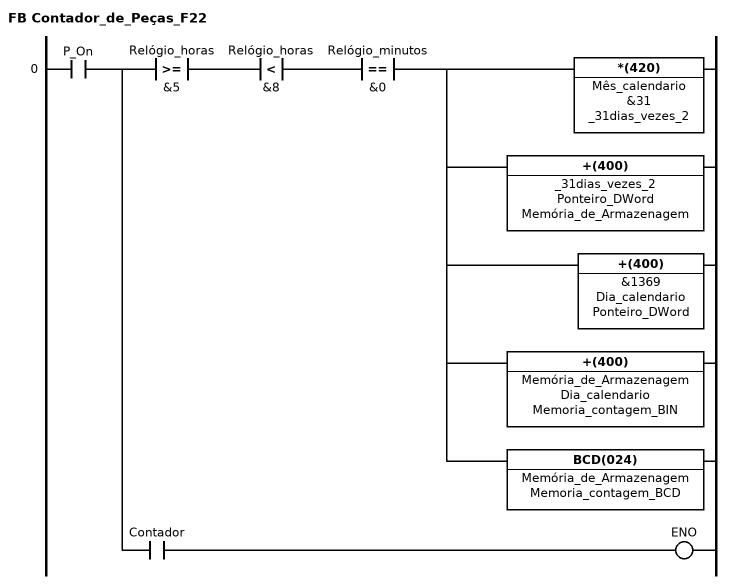
; rung 0
LD P_On
OUT TR0
AND>=(325) Relógio_horas &5
AND<(310) Relógio_horas &8
AND=(300) Relógio_minutos &0
*(420) Mês_calendario &31 _31dias_vezes_2
+(400) _31dias_vezes_2 Ponteiro_DWord Memória_de_Armazenagem
+(400) &1369 Dia_calendario Ponteiro_DWord
+(400) Memória_de_Armazenagem Dia_calendario Memoria_contagem_BIN
BCD(024) Memória_de_Armazenagem Memoria_contagem_BCD
LD TR0
AND Contador
OUT ENO

## Function block Contador_de_Peças_RC41
VAR_INPUT
  Relógio_horas : WORD;
  Relógio_minutos : WORD;
  Dia_calendario : WORD;
  Mês_calendario : WORD;
  Contador : BOOL;
END_VAR
VAR
  _31dias_vezes_2 AT D520 : WORD;
  Ponteiro_DWord AT D522 : WORD;
  Memória_de_Armazenagem AT D524 : WORD;
  Memoria_contagem_BIN AT D526 : WORD;
  Memoria_contagem_BCD AT D528 : WORD;
END_VAR

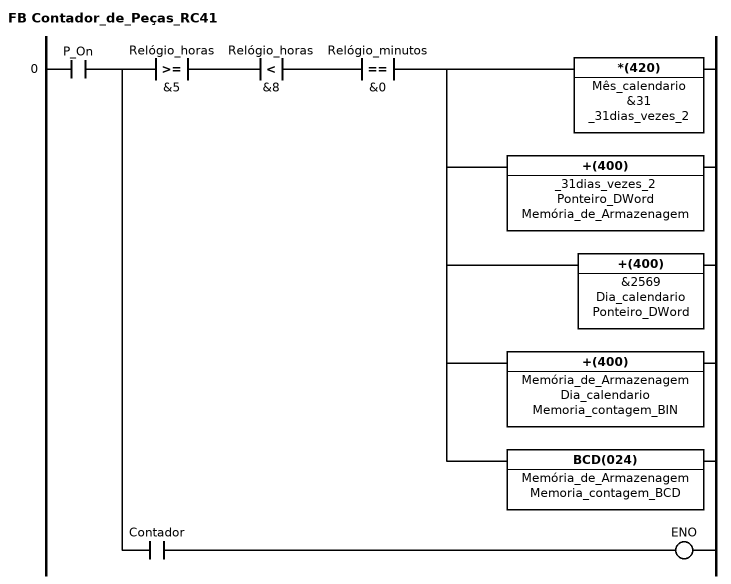
; rung 0
LD P_On
OUT TR0
AND>=(325) Relógio_horas &5
AND<(310) Relógio_horas &8
AND=(300) Relógio_minutos &0
*(420) Mês_calendario &31 _31dias_vezes_2
+(400) _31dias_vezes_2 Ponteiro_DWord Memória_de_Armazenagem
+(400) &2569 Dia_calendario Ponteiro_DWord
+(400) Memória_de_Armazenagem Dia_calendario Memoria_contagem_BIN
BCD(024) Memória_de_Armazenagem Memoria_contagem_BCD
LD TR0
AND Contador
OUT ENO

## Function block Contador_de_Peças_RC42
VAR_INPUT
  Relógio_horas : WORD;
  Relógio_minutos : WORD;
  Dia_calendario : WORD;
  Mês_calendario : WORD;
  Contador : BOOL;
END_VAR
VAR
  _31dias_vezes_2 AT D540 : WORD;
  Ponteiro_DWord AT D542 : WORD;
  Memória_de_Armazenagem AT D544 : WORD;
  Memoria_contagem_BIN AT D546 : WORD;
  Memoria_contagem_BCD AT D548 : WORD;
END_VAR

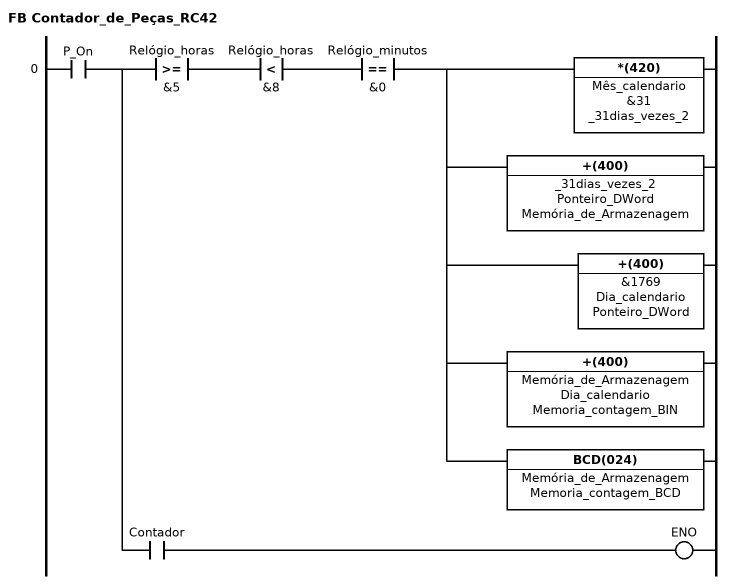
; rung 0
LD P_On
OUT TR0
AND>=(325) Relógio_horas &5
AND<(310) Relógio_horas &8
AND=(300) Relógio_minutos &0
*(420) Mês_calendario &31 _31dias_vezes_2
+(400) _31dias_vezes_2 Ponteiro_DWord Memória_de_Armazenagem
+(400) &1769 Dia_calendario Ponteiro_DWord
+(400) Memória_de_Armazenagem Dia_calendario Memoria_contagem_BIN
BCD(024) Memória_de_Armazenagem Memoria_contagem_BCD
LD TR0
AND Contador
OUT ENO

## Function block Contador_de_Peças_RC43
VAR_INPUT
  Relógio_horas : WORD;
  Relógio_minutos : WORD;
  Dia_calendario : WORD;
  Mês_calendario : WORD;
  Contador : BOOL;
END_VAR
VAR
  _31dias_vezes_2 AT D500 : WORD;
  Ponteiro_DWord AT D502 : WORD;
  Memória_de_Armazenagem AT D504 : WORD;
  Memoria_contagem_BIN AT D506 : WORD;
  Memoria_contagem_BCD AT D508 : WORD;
END_VAR

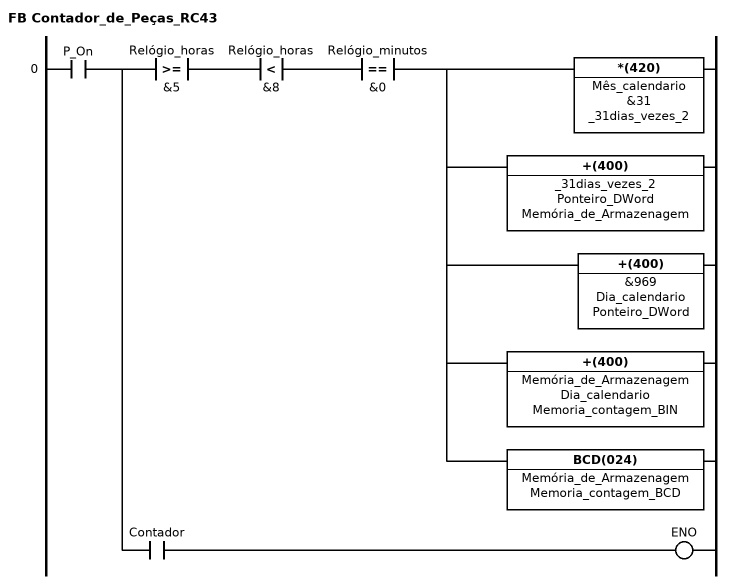
; rung 0
LD P_On
OUT TR0
AND>=(325) Relógio_horas &5
AND<(310) Relógio_horas &8
AND=(300) Relógio_minutos &0
*(420) Mês_calendario &31 _31dias_vezes_2
+(400) _31dias_vezes_2 Ponteiro_DWord Memória_de_Armazenagem
+(400) &969 Dia_calendario Ponteiro_DWord
+(400) Memória_de_Armazenagem Dia_calendario Memoria_contagem_BIN
BCD(024) Memória_de_Armazenagem Memoria_contagem_BCD
LD TR0
AND Contador
OUT ENO